{attribute 'strict'}
TYPE E_KR_AutoExtState :
(
    Idle := 0,

    CheckReady,
    MoveEnableOn,
    DrivesOnPulse,
    WaitDrivesReady,

    WaitPgnoReq,
    RetryDrivesOnPulse,

    SetProgramNo,
    ExtStartPulse,
    WaitProgramActive,

    Running,
    Finish,

    Error
);
END_TYPE

(* stored: Version 1.1.0.1, ProductVersion 3.1.4024.16
   DUT E_KR_AutoExtState: Id {bd7e0e08-0eed-4ada-a2a4-61f0381499e5} *)
